// Mitsubishi GX Works2 project: 02.CumLongVo   PLC: FX3U/FX3UC

// global labels: Positon
VAR_GLOBAL
  Ser_Org : BOOL;
  Ser_Home_Done : BOOL;
  A_M : BOOL;
  Emer : BOOL;
  ON_ABS : BOOL;
  Pos_Tag_ABS : DINT;  (* mm *)
  Speed_Tag_ABS : DINT;  (* mm/s *)
  Excute_ABS : BOOL;
END_VAR

// global labels: Pro_Con_TF_J
VAR_GLOBAL
  Rev_J_Done : BOOL;
  Pro_Rev_J : BOOL;
  Req_Cov_W_Rev : BOOL;
  Conv_TF_J_Ready : BOOL;
  D_Step3_TF_Frame : TIMER;
  Cf_Install_Frame : BOOL;
END_VAR

// global labels: Pro_Con_Wait
VAR_GLOBAL
  Conv_W_Ready : BOOL;
  Conv_W_Rev_Done : BOOL;
  Req_Clus_Ep_Rev : BOOL;
  D_Req_ClusEp_Rev : TIMER;
END_VAR

// global labels: Cluster_BT
VAR_GLOBAL
  BT_Req_Rev_J : BOOL;
END_VAR

// global labels: Pro_Clus_Ep
VAR_GLOBAL
  Clus_Ep_Ready_Rev : BOOL;
  Clus_Ep_Rev_Done : BOOL;
  Req_Con_Out_Rev : BOOL;
  Clus_Ep_Safety : BOOL;
  Ex_Ep_Frame : BOOL;
  Stp_Ep_Fr : INT;
  Pos_Saf : REAL;
  Pos_Kep : REAL;
  Pos_Ep : REAL;
  Pos_Tar : REAL;
  Ep_Done : BOOL;
  Pos_Safe_Cyl_DT : REAL;
END_VAR

// global labels: Pro_Conv_Out
VAR_GLOBAL
  Conv_Out_Ready_Rev : BOOL;
  Conv_Out_Rev_Done : BOOL;
  Req_Clus_Drill_Rev : BOOL;
  TimeOut_BT : TIMER;
  Stp_Measuse : INT;
  T_Val_Err_Ams : REAL;
  Val_Err_Ams : REAL;
  Result : INT;
  D_Measure : TIMER;
  Stp_Rev_Conv_Out : BOOL;
  Measure_Done : BOOL;
  D_Conv_Out_Ready : TIMER;
  Standar_P : REAL;
  Standar_N : REAL;
  Value_1 : REAL;
  Value_2 : REAL;
  Value_Temp : REAL;
  D_Value2 : TIMER;
  Value_TempOut : REAL;
  O_Val_Err_Ams : REAL;
END_VAR

// global labels: TF_Jig
VAR_GLOBAL
  Step_TF_J : INT;
  Ex_TF_J : BOOL;
  Done_TF_J : BOOL;
  D_Done_J : TIMER;
END_VAR

// global labels: Clus_Drill
VAR_GLOBAL
  Clus_Drill_Ready_Rev : BOOL;
END_VAR

// global labels: Pro_Clus_TF_Frame
VAR_GLOBAL
  Clus_Cyl_TF_Frame_Ready : BOOL;  (* Ready *)
  Ex_TF_Frame : BOOL;
  D_Noti_Ex_Ep : TIMER;
  D_Nha_Kep1 : TIMER;
  D_PickDone : TIMER;
  Skip_Heater : BOOL;
  Stp_TF_Fr : INT;
  Clus_TF_Frame_Safety : BOOL;
  Ready_TF_Frame : BOOL;
  TF_Frame_Safe_Ep : BOOL;
  TF_Fr_Codition_TF_J : BOOL;
END_VAR

// global labels: Pro_Heater
VAR_GLOBAL
  Ex_Heater : BOOL;
  Heater_Done : BOOL;
  Heater_Busy : BOOL;
  Heater_Ready : BOOL;
  Heater_Safety : BOOL;
  Stp_Heater : INT;
  T_Target : REAL;
  Pre_Heater : BOOL;
END_VAR

PROGRAM Main
VAR
  Conv_TF_J : Conv_TF_J;
  Conv_Wait : Conv_Wait;
  C_Cyl_TF_J : C_Cyl_TF_J;
  C_Cyl_TF_SP : C_Cyl_TF_SP;
  Heater : Heater;
  Conv_Out : Conv_Out;
  Ctr_Mc : Ctr_MC;
  C_Shell : C_ShellCage;
END_VAR
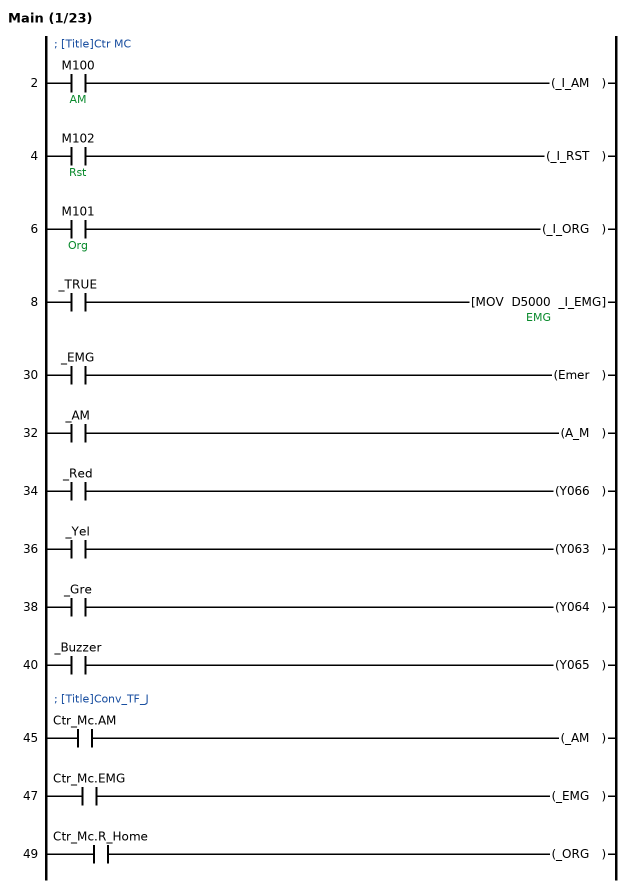
; FB BLK START Ctr_MC(Ctr_Mc)
; [Title]Ctr MC
2     LD      M100  ; AM
      OUT     _I_AM
4     LD      M102  ; Rst
      OUT     _I_RST
6     LD      M101  ; Org
      OUT     _I_ORG
8     LD      _TRUE
      MOV     D5000 _I_EMG  ; EMG
; FB START
; FB_NAME Ctr_MC
; INSTANCE_NAME Ctr_Mc
; FB IN_B:I_AM
; FB OUT_Flag_Run:B
; FB IN_B:I_RST
; FB OUT_EMG:B
; FB IN_B:I_ORG
; FB OUT_AM:B
; FB IN_W:I_EMG
; FB OUT_R_Home:B
; FB OUT_Red:B
; FB OUT_Yel:B
; FB OUT_Gre:B
; FB OUT_Buzzer:B
; FB END
30    LD      _EMG
      OUT     Emer
32    LD      _AM
      OUT     A_M
34    LD      _Red
      OUT     Y066
36    LD      _Yel
      OUT     Y063
38    LD      _Gre
      OUT     Y064
40    LD      _Buzzer
      OUT     Y065
; FB BLK END
; FB BLK START Conv_TF_J(Conv_TF_J)
; [Title]Conv_TF_J
45    LD      Ctr_Mc.AM
      OUT     _AM
47    LD      Ctr_Mc.EMG
      OUT     _EMG
49    LD      Ctr_Mc.R_Home
      OUT     _ORG
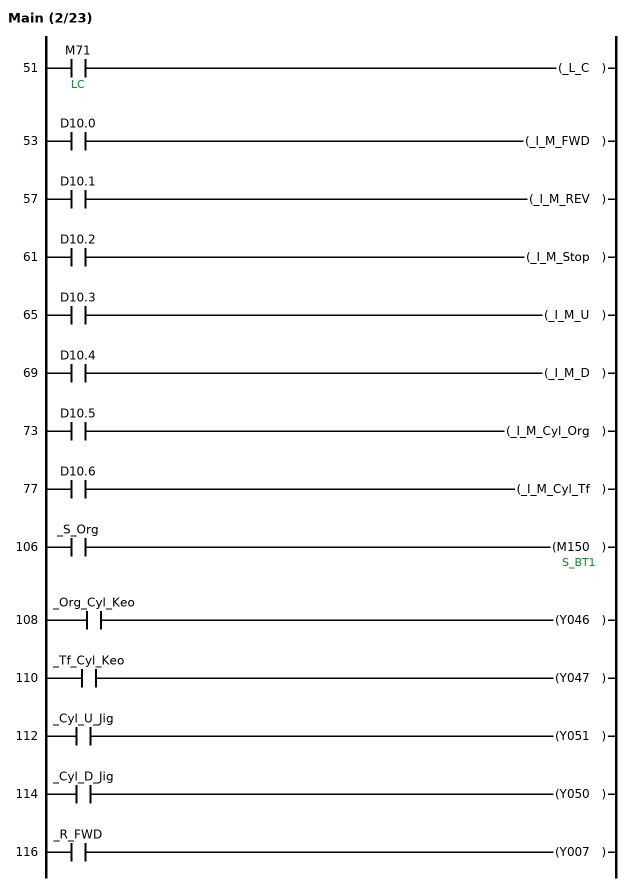
51    LD      M71  ; LC
      OUT     _L_C
53    LD      D10.0
      OUT     _I_M_FWD
57    LD      D10.1
      OUT     _I_M_REV
61    LD      D10.2
      OUT     _I_M_Stop
65    LD      D10.3
      OUT     _I_M_U
69    LD      D10.4
      OUT     _I_M_D
73    LD      D10.5
      OUT     _I_M_Cyl_Org
77    LD      D10.6
      OUT     _I_M_Cyl_Tf
; FB START
; FB_NAME Conv_TF_J
; INSTANCE_NAME Conv_TF_J
; FB IN_B:AM
; FB OUT_S_Org:B
; FB IN_B:EMG
; FB OUT_Org_Cyl_Keo:B
; FB IN_B:ORG
; FB OUT_Tf_Cyl_Keo:B
; FB IN_B:L_C
; FB OUT_Cyl_U_Jig:B
; FB IN_B:I_M_FWD
; FB OUT_Cyl_D_Jig:B
; FB IN_B:I_M_REV
; FB OUT_R_FWD:B
; FB IN_B:I_M_Stop
; FB OUT_R_REV:B
; FB IN_B:I_M_U
; FB IN_B:I_M_D
; FB IN_B:I_M_Cyl_Org
; FB IN_B:I_M_Cyl_Tf
; FB IN_W:A_S_Cyl_UD
; FB IN_W:A_S_Cyl_Tf
; FB IN_W:A_S_Conv
; FB END
106   LD      _S_Org
      OUT     M150  ; S_BT1
108   LD      _Org_Cyl_Keo
      OUT     Y046
110   LD      _Tf_Cyl_Keo
      OUT     Y047
112   LD      _Cyl_U_Jig
      OUT     Y051
114   LD      _Cyl_D_Jig
      OUT     Y050
116   LD      _R_FWD
      OUT     Y007
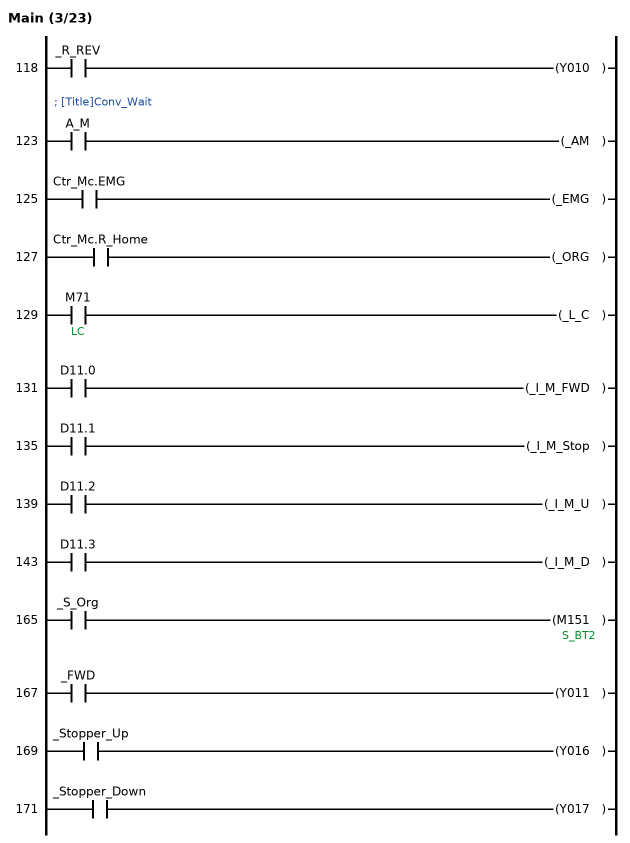
118   LD      _R_REV
      OUT     Y010
; FB BLK END
; FB BLK START Conv_Wait(Conv_Wait)
; [Title]Conv_Wait
123   LD      A_M
      OUT     _AM
125   LD      Ctr_Mc.EMG
      OUT     _EMG
127   LD      Ctr_Mc.R_Home
      OUT     _ORG
129   LD      M71  ; LC
      OUT     _L_C
131   LD      D11.0
      OUT     _I_M_FWD
135   LD      D11.1
      OUT     _I_M_Stop
139   LD      D11.2
      OUT     _I_M_U
143   LD      D11.3
      OUT     _I_M_D
; FB START
; FB_NAME Conv_Wait
; INSTANCE_NAME Conv_Wait
; FB IN_B:AM
; FB OUT_S_Org:B
; FB IN_B:EMG
; FB OUT_FWD:B
; FB IN_B:ORG
; FB OUT_Stopper_Up:B
; FB IN_B:L_C
; FB OUT_Stopper_Down:B
; FB IN_B:I_M_FWD
; FB IN_B:I_M_Stop
; FB IN_B:I_M_U
; FB IN_B:I_M_D
; FB IN_B:A_FWD
; FB IN_W:A_S_Stp
; FB END
165   LD      _S_Org
      OUT     M151  ; S_BT2
167   LD      _FWD
      OUT     Y011
169   LD      _Stopper_Up
      OUT     Y016
171   LD      _Stopper_Down
      OUT     Y017
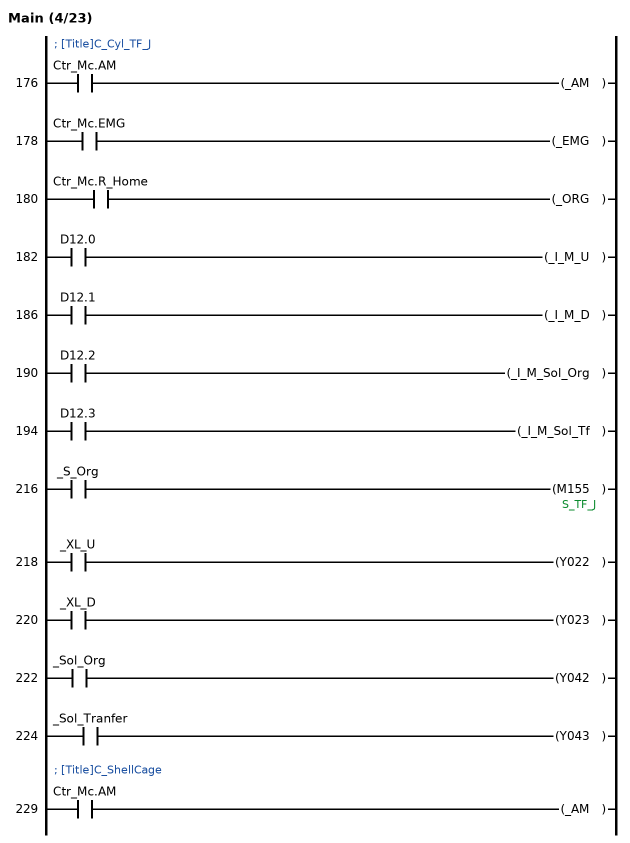
; FB BLK END
; FB BLK START C_Cyl_TF_J(C_Cyl_TF_J)
; [Title]C_Cyl_TF_J
176   LD      Ctr_Mc.AM
      OUT     _AM
178   LD      Ctr_Mc.EMG
      OUT     _EMG
180   LD      Ctr_Mc.R_Home
      OUT     _ORG
182   LD      D12.0
      OUT     _I_M_U
186   LD      D12.1
      OUT     _I_M_D
190   LD      D12.2
      OUT     _I_M_Sol_Org
194   LD      D12.3
      OUT     _I_M_Sol_Tf
; FB START
; FB_NAME C_Cyl_TF_J
; INSTANCE_NAME C_Cyl_TF_J
; FB IN_B:AM
; FB OUT_S_Org:B
; FB IN_B:EMG
; FB OUT_XL_U:B
; FB IN_B:ORG
; FB OUT_XL_D:B
; FB IN_B:I_M_U
; FB OUT_Sol_Org:B
; FB IN_B:I_M_D
; FB OUT_Sol_Tranfer:B
; FB IN_B:I_M_Sol_Org
; FB IN_B:I_M_Sol_Tf
; FB IN_W:A_Status_XL_U
; FB IN_W:A_S_Cyl_Tf
; FB END
216   LD      _S_Org
      OUT     M155  ; S_TF_J
218   LD      _XL_U
      OUT     Y022
220   LD      _XL_D
      OUT     Y023
222   LD      _Sol_Org
      OUT     Y042
224   LD      _Sol_Tranfer
      OUT     Y043
; FB BLK END
; FB BLK START C_ShellCage(C_Shell)
; [Title]C_ShellCage
229   LD      Ctr_Mc.AM
      OUT     _AM
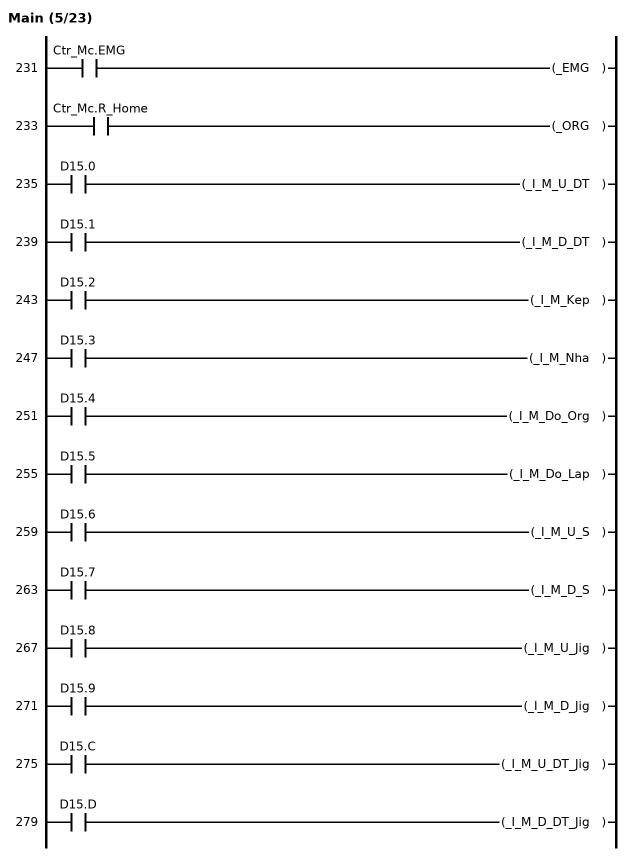
231   LD      Ctr_Mc.EMG
      OUT     _EMG
233   LD      Ctr_Mc.R_Home
      OUT     _ORG
235   LD      D15.0
      OUT     _I_M_U_DT
239   LD      D15.1
      OUT     _I_M_D_DT
243   LD      D15.2
      OUT     _I_M_Kep
247   LD      D15.3
      OUT     _I_M_Nha
251   LD      D15.4
      OUT     _I_M_Do_Org
255   LD      D15.5
      OUT     _I_M_Do_Lap
259   LD      D15.6
      OUT     _I_M_U_S
263   LD      D15.7
      OUT     _I_M_D_S
267   LD      D15.8
      OUT     _I_M_U_Jig
271   LD      D15.9
      OUT     _I_M_D_Jig
275   LD      D15.C
      OUT     _I_M_U_DT_Jig
279   LD      D15.D
      OUT     _I_M_D_DT_Jig
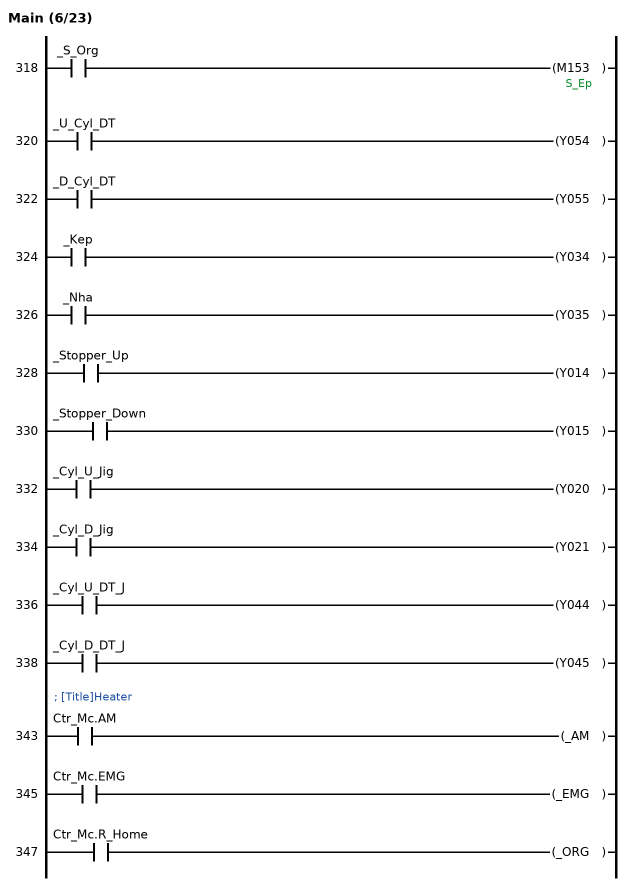
; FB START
; FB_NAME C_ShellCage
; INSTANCE_NAME C_Shell
; FB IN_B:AM
; FB OUT_S_Org:B
; FB IN_B:EMG
; FB OUT_U_Cyl_DT:B
; FB IN_B:ORG
; FB OUT_D_Cyl_DT:B
; FB IN_B:I_M_U_DT
; FB OUT_Kep:B
; FB IN_B:I_M_D_DT
; FB OUT_Nha:B
; FB IN_B:I_M_Kep
; FB OUT_Stopper_Up:B
; FB IN_B:I_M_Nha
; FB OUT_Stopper_Down:B
; FB IN_B:I_M_Do_Org
; FB OUT_Cyl_U_Jig:B
; FB IN_B:I_M_Do_Lap
; FB OUT_Cyl_D_Jig:B
; FB IN_B:I_M_U_S
; FB OUT_Cyl_U_DT_J:B
; FB IN_B:I_M_D_S
; FB OUT_Cyl_D_DT_J:B
; FB IN_B:I_M_U_Jig
; FB IN_B:I_M_D_Jig
; FB IN_B:I_M_U_DT_Jig
; FB IN_B:I_M_D_DT_Jig
; FB IN_W:A_S_Cyl_DT
; FB IN_W:A_S_Cyl_Kep
; FB IN_W:A_S_Stp
; FB IN_W:A_S_UD_J
; FB IN_W:A_S_DT_J
; FB END
318   LD      _S_Org
      OUT     M153  ; S_Ep
320   LD      _U_Cyl_DT
      OUT     Y054
322   LD      _D_Cyl_DT
      OUT     Y055
324   LD      _Kep
      OUT     Y034
326   LD      _Nha
      OUT     Y035
328   LD      _Stopper_Up
      OUT     Y014
330   LD      _Stopper_Down
      OUT     Y015
332   LD      _Cyl_U_Jig
      OUT     Y020
334   LD      _Cyl_D_Jig
      OUT     Y021
336   LD      _Cyl_U_DT_J
      OUT     Y044
338   LD      _Cyl_D_DT_J
      OUT     Y045
; FB BLK END
; FB BLK START Heater(Heater)
; [Title]Heater
343   LD      Ctr_Mc.AM
      OUT     _AM
345   LD      Ctr_Mc.EMG
      OUT     _EMG
347   LD      Ctr_Mc.R_Home
      OUT     _ORG
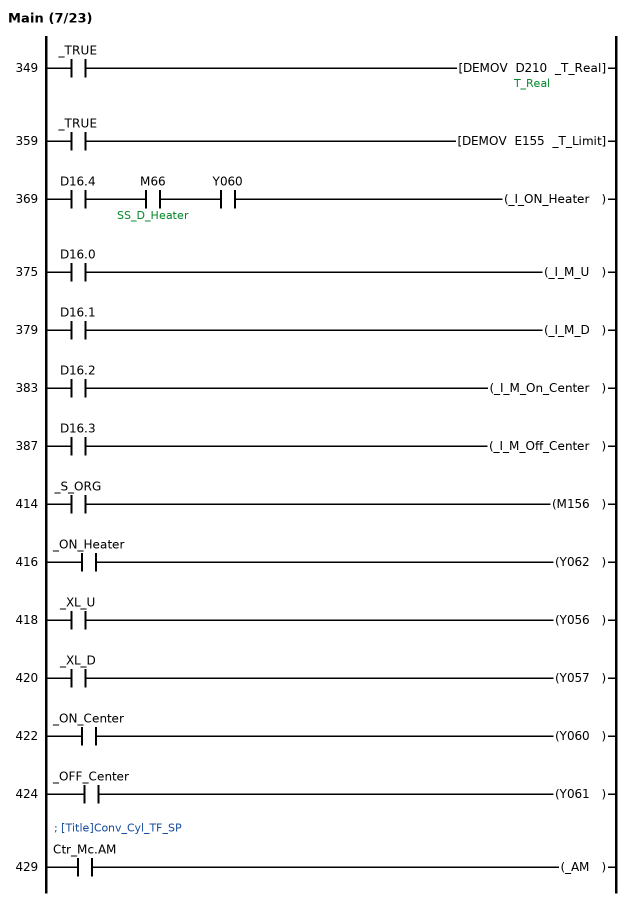
349   LD      _TRUE
      DEMOV   D210 _T_Real  ; T_Real
359   LD      _TRUE
      DEMOV   E155 _T_Limit
369   LD      D16.4
      AND     M66  ; SS_D_Heater
      AND     Y060
      OUT     _I_ON_Heater
375   LD      D16.0
      OUT     _I_M_U
379   LD      D16.1
      OUT     _I_M_D
383   LD      D16.2
      OUT     _I_M_On_Center
387   LD      D16.3
      OUT     _I_M_Off_Center
; FB START
; FB_NAME Heater
; INSTANCE_NAME Heater
; FB IN_B:AM
; FB OUT_S_ORG:B
; FB IN_B:EMG
; FB OUT_ON_Heater:B
; FB IN_B:ORG
; FB OUT_XL_U:B
; FB IN_E:T_Real
; FB OUT_XL_D:B
; FB IN_E:T_Limit
; FB OUT_ON_Center:B
; FB IN_B:I_ON_Heater
; FB OUT_OFF_Center:B
; FB IN_B:I_M_U
; FB IN_B:I_M_D
; FB IN_B:I_M_On_Center
; FB IN_B:I_M_Off_Center
; FB IN_B:A_ON_Heater
; FB IN_W:A_S_Cyl_UD
; FB IN_W:A_Status_Center
; FB END
414   LD      _S_ORG
      OUT     M156
416   LD      _ON_Heater
      OUT     Y062
418   LD      _XL_U
      OUT     Y056
420   LD      _XL_D
      OUT     Y057
422   LD      _ON_Center
      OUT     Y060
424   LD      _OFF_Center
      OUT     Y061
; FB BLK END
; FB BLK START C_Cyl_TF_SP(C_Cyl_TF_SP)
; [Title]Conv_Cyl_TF_SP
429   LD      Ctr_Mc.AM
      OUT     _AM
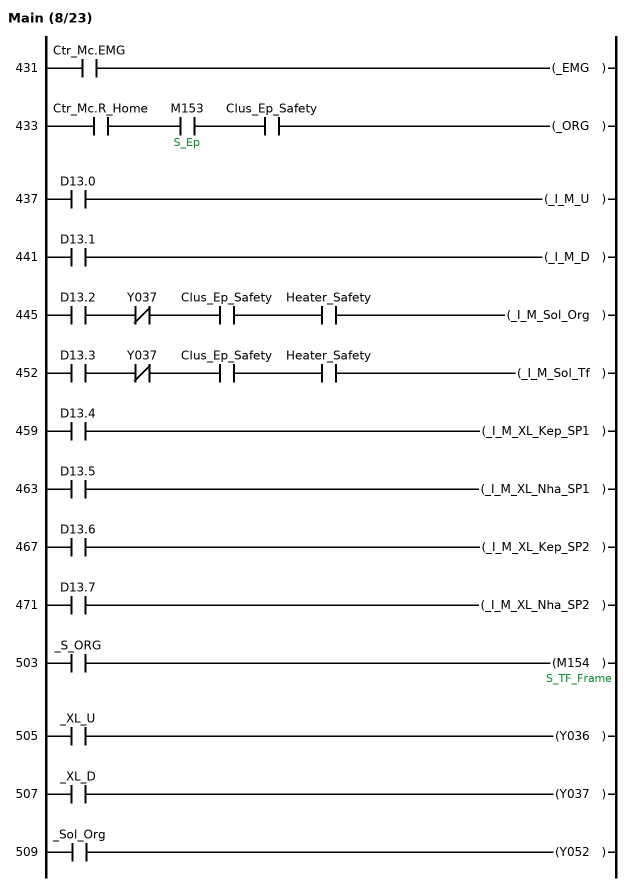
431   LD      Ctr_Mc.EMG
      OUT     _EMG
433   LD      Ctr_Mc.R_Home
      AND     M153  ; S_Ep
      AND     Clus_Ep_Safety
      OUT     _ORG
437   LD      D13.0
      OUT     _I_M_U
441   LD      D13.1
      OUT     _I_M_D
445   LD      D13.2
      ANI     Y037
      AND     Clus_Ep_Safety
      AND     Heater_Safety
      OUT     _I_M_Sol_Org
452   LD      D13.3
      ANI     Y037
      AND     Clus_Ep_Safety
      AND     Heater_Safety
      OUT     _I_M_Sol_Tf
459   LD      D13.4
      OUT     _I_M_XL_Kep_SP1
463   LD      D13.5
      OUT     _I_M_XL_Nha_SP1
467   LD      D13.6
      OUT     _I_M_XL_Kep_SP2
471   LD      D13.7
      OUT     _I_M_XL_Nha_SP2
; FB START
; FB_NAME C_Cyl_TF_SP
; INSTANCE_NAME C_Cyl_TF_SP
; FB IN_B:AM
; FB OUT_S_ORG:B
; FB IN_B:EMG
; FB OUT_XL_U:B
; FB IN_B:ORG
; FB OUT_XL_D:B
; FB IN_B:I_M_U
; FB OUT_Sol_Org:B
; FB IN_B:I_M_D
; FB OUT_Sol_Tranfer:B
; FB IN_B:I_M_Sol_Org
; FB OUT_XL_Kep_SP1:B
; FB IN_B:I_M_Sol_Tf
; FB OUT_XL_Mo_SP1:B
; FB IN_B:I_M_XL_Kep_SP1
; FB OUT_XL_Kep_SP2:B
; FB IN_B:I_M_XL_Nha_SP1
; FB OUT_XL_Mo_SP2:B
; FB IN_B:I_M_XL_Kep_SP2
; FB IN_B:I_M_XL_Nha_SP2
; FB IN_W:A_Status_XL_U
; FB IN_W:A_S_Cyl_Tf
; FB IN_W:A_S_Cyl_Kep_1
; FB IN_W:A_S_Cyl_Kep_2
; FB END
503   LD      _S_ORG
      OUT     M154  ; S_TF_Frame
505   LD      _XL_U
      OUT     Y036
507   LD      _XL_D
      OUT     Y037
509   LD      _Sol_Org
      OUT     Y052
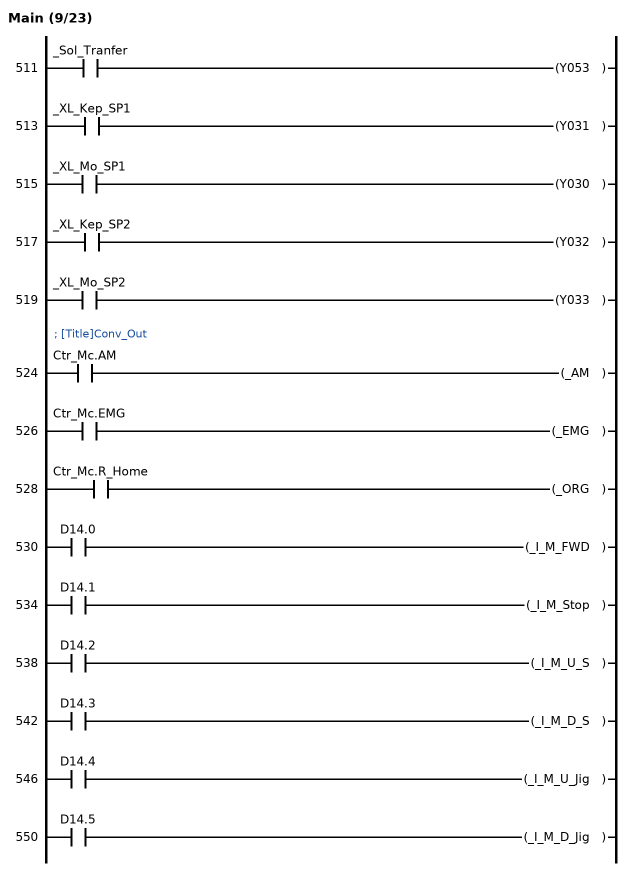
511   LD      _Sol_Tranfer
      OUT     Y053
513   LD      _XL_Kep_SP1
      OUT     Y031
515   LD      _XL_Mo_SP1
      OUT     Y030
517   LD      _XL_Kep_SP2
      OUT     Y032
519   LD      _XL_Mo_SP2
      OUT     Y033
; FB BLK END
; FB BLK START Conv_Out(Conv_Out)
; [Title]Conv_Out
524   LD      Ctr_Mc.AM
      OUT     _AM
526   LD      Ctr_Mc.EMG
      OUT     _EMG
528   LD      Ctr_Mc.R_Home
      OUT     _ORG
530   LD      D14.0
      OUT     _I_M_FWD
534   LD      D14.1
      OUT     _I_M_Stop
538   LD      D14.2
      OUT     _I_M_U_S
542   LD      D14.3
      OUT     _I_M_D_S
546   LD      D14.4
      OUT     _I_M_U_Jig
550   LD      D14.5
      OUT     _I_M_D_Jig
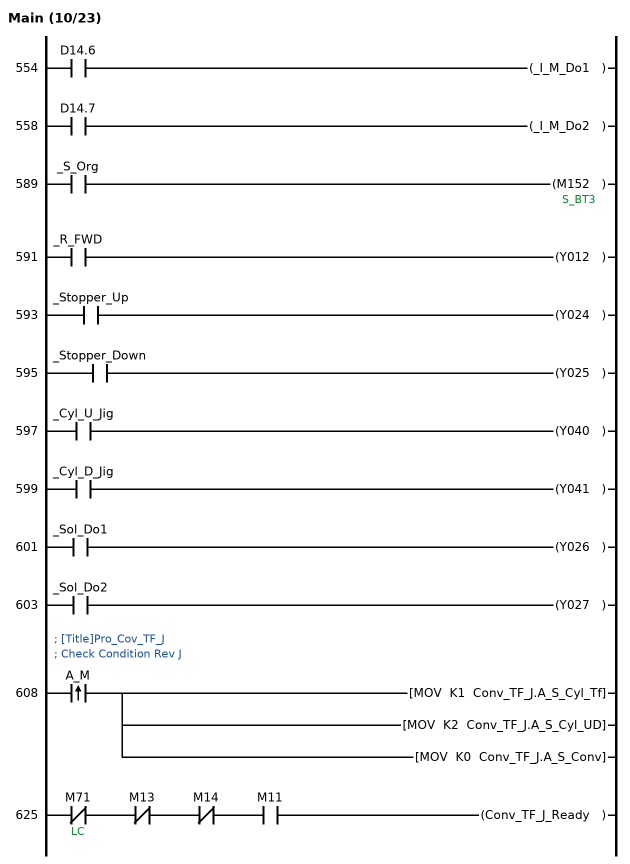
554   LD      D14.6
      OUT     _I_M_Do1
558   LD      D14.7
      OUT     _I_M_Do2
; FB START
; FB_NAME Conv_Out
; INSTANCE_NAME Conv_Out
; FB IN_B:AM
; FB OUT_S_Org:B
; FB IN_B:EMG
; FB OUT_R_FWD:B
; FB IN_B:ORG
; FB OUT_Stopper_Up:B
; FB IN_B:I_M_FWD
; FB OUT_Stopper_Down:B
; FB IN_B:I_M_Stop
; FB OUT_Cyl_U_Jig:B
; FB IN_B:I_M_U_S
; FB OUT_Cyl_D_Jig:B
; FB IN_B:I_M_D_S
; FB OUT_Sol_Do1:B
; FB IN_B:I_M_U_Jig
; FB OUT_Sol_Do2:B
; FB IN_B:I_M_D_Jig
; FB IN_B:I_M_Do1
; FB IN_B:I_M_Do2
; FB IN_W:A_S_Cyl_UD
; FB IN_W:A_S_Stp
; FB IN_B:A_FWD
; FB IN_W:A_S_Do
; FB END
589   LD      _S_Org
      OUT     M152  ; S_BT3
591   LD      _R_FWD
      OUT     Y012
593   LD      _Stopper_Up
      OUT     Y024
595   LD      _Stopper_Down
      OUT     Y025
597   LD      _Cyl_U_Jig
      OUT     Y040
599   LD      _Cyl_D_Jig
      OUT     Y041
601   LD      _Sol_Do1
      OUT     Y026
603   LD      _Sol_Do2
      OUT     Y027
; FB BLK END
; [Title]Pro_Cov_TF_J
; Check Condition Rev J
608   LDP     A_M
      MOV     K1 Conv_TF_J.A_S_Cyl_Tf
      MOV     K2 Conv_TF_J.A_S_Cyl_UD
      MOV     K0 Conv_TF_J.A_S_Conv
625   LDI     M71  ; LC
      ANI     M13
      ANI     M14
      AND     M11
      OUT     Conv_TF_J_Ready
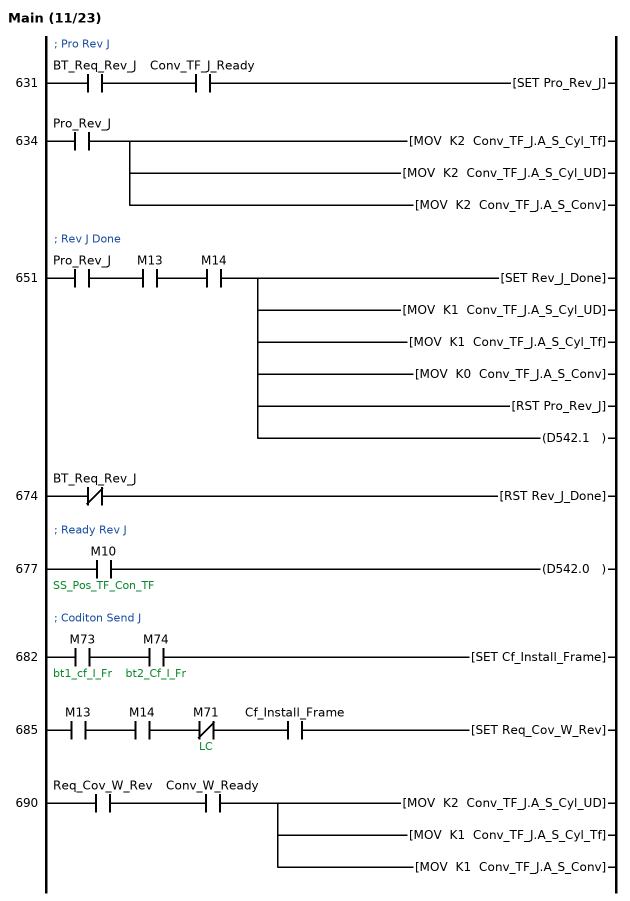
; Pro Rev J
631   LD      BT_Req_Rev_J
      AND     Conv_TF_J_Ready
      SET     Pro_Rev_J
634   LD      Pro_Rev_J
      MOV     K2 Conv_TF_J.A_S_Cyl_Tf
      MOV     K2 Conv_TF_J.A_S_Cyl_UD
      MOV     K2 Conv_TF_J.A_S_Conv
; Rev J Done
651   LD      Pro_Rev_J
      AND     M13
      AND     M14
      SET     Rev_J_Done
      MOV     K1 Conv_TF_J.A_S_Cyl_UD
      MOV     K1 Conv_TF_J.A_S_Cyl_Tf
      MOV     K0 Conv_TF_J.A_S_Conv
      RST     Pro_Rev_J
      OUT     D542.1
674   LDI     BT_Req_Rev_J
      RST     Rev_J_Done
; Ready Rev J
677   LD      M10  ; SS_Pos_TF_Con_TF
      OUT     D542.0
; Coditon Send J
682   LD      M73  ; bt1_cf_I_Fr
      AND     M74  ; bt2_Cf_I_Fr
      SET     Cf_Install_Frame
685   LD      M13
      AND     M14
      ANI     M71  ; LC
      AND     Cf_Install_Frame
      SET     Req_Cov_W_Rev
690   LD      Req_Cov_W_Rev
      AND     Conv_W_Ready
      MOV     K2 Conv_TF_J.A_S_Cyl_UD
      MOV     K1 Conv_TF_J.A_S_Cyl_Tf
      MOV     K1 Conv_TF_J.A_S_Conv
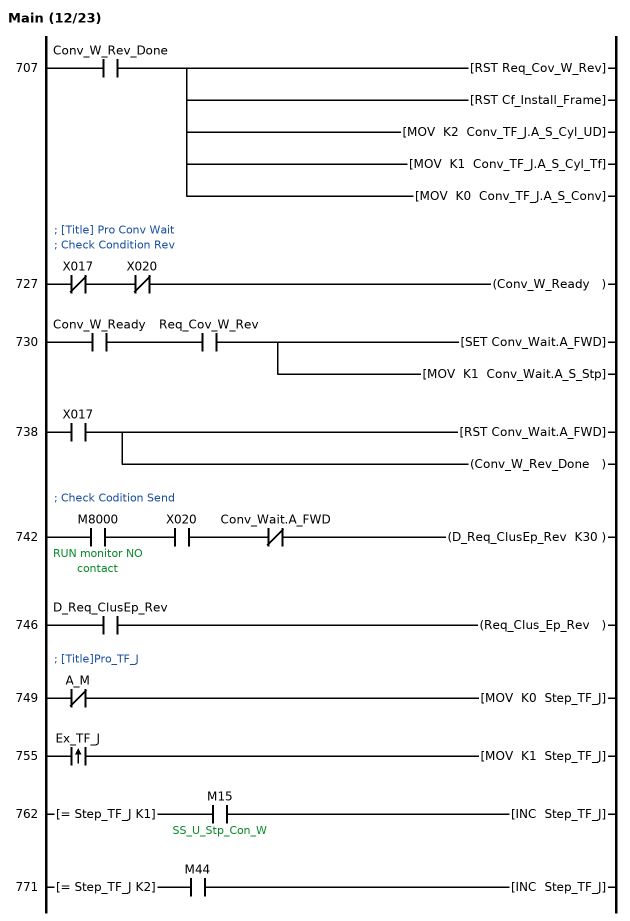
707   LD      Conv_W_Rev_Done
      RST     Req_Cov_W_Rev
      RST     Cf_Install_Frame
      MOV     K2 Conv_TF_J.A_S_Cyl_UD
      MOV     K1 Conv_TF_J.A_S_Cyl_Tf
      MOV     K0 Conv_TF_J.A_S_Conv
; [Title] Pro Conv Wait
; Check Condition Rev
727   LDI     X017
      ANI     X020
      OUT     Conv_W_Ready
730   LD      Conv_W_Ready
      AND     Req_Cov_W_Rev
      SET     Conv_Wait.A_FWD
      MOV     K1 Conv_Wait.A_S_Stp
738   LD      X017
      RST     Conv_Wait.A_FWD
      OUT     Conv_W_Rev_Done
; Check Codition Send
742   LD      M8000  ; RUN monitor NO contact
      AND     X020
      ANI     Conv_Wait.A_FWD
      OUT     D_Req_ClusEp_Rev K30
746   LD      D_Req_ClusEp_Rev
      OUT     Req_Clus_Ep_Rev
; [Title]Pro_TF_J
749   LDI     A_M
      MOV     K0 Step_TF_J
755   LDP     Ex_TF_J
      MOV     K1 Step_TF_J
762   LD=     Step_TF_J K1
      AND     M15  ; SS_U_Stp_Con_W
      INC     Step_TF_J
771   LD=     Step_TF_J K2
      AND     M44
      INC     Step_TF_J
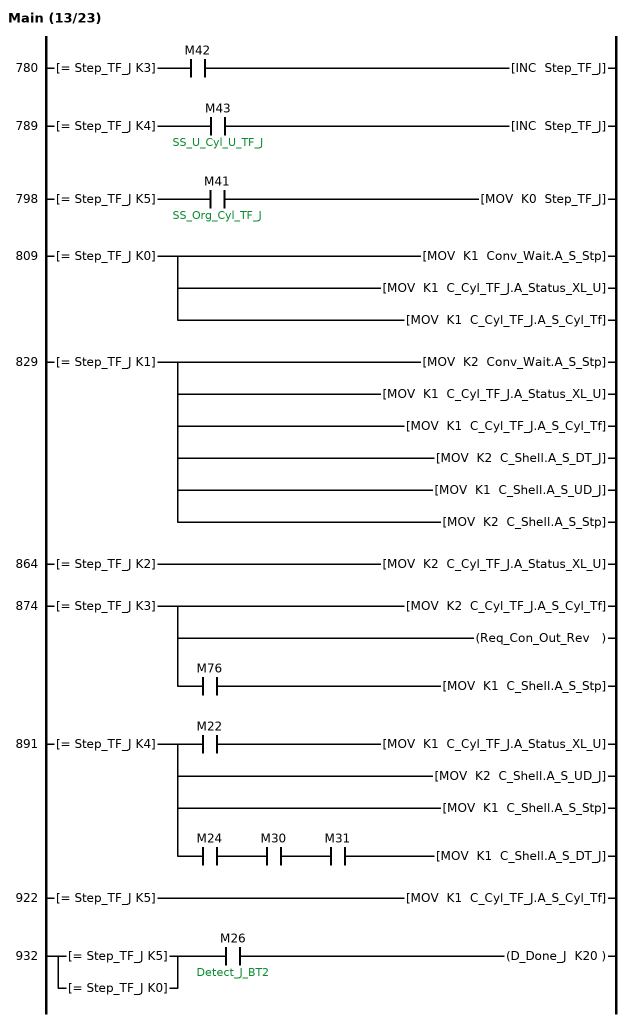
780   LD=     Step_TF_J K3
      AND     M42
      INC     Step_TF_J
789   LD=     Step_TF_J K4
      AND     M43  ; SS_U_Cyl_U_TF_J
      INC     Step_TF_J
798   LD=     Step_TF_J K5
      AND     M41  ; SS_Org_Cyl_TF_J
      MOV     K0 Step_TF_J
809   LD=     Step_TF_J K0
      MOV     K1 Conv_Wait.A_S_Stp
      MOV     K1 C_Cyl_TF_J.A_Status_XL_U
      MOV     K1 C_Cyl_TF_J.A_S_Cyl_Tf
829   LD=     Step_TF_J K1
      MOV     K2 Conv_Wait.A_S_Stp
      MOV     K1 C_Cyl_TF_J.A_Status_XL_U
      MOV     K1 C_Cyl_TF_J.A_S_Cyl_Tf
      MOV     K2 C_Shell.A_S_DT_J
      MOV     K1 C_Shell.A_S_UD_J
      MOV     K2 C_Shell.A_S_Stp
864   LD=     Step_TF_J K2
      MOV     K2 C_Cyl_TF_J.A_Status_XL_U
874   LD=     Step_TF_J K3
      MOV     K2 C_Cyl_TF_J.A_S_Cyl_Tf
      OUT     Req_Con_Out_Rev
      AND     M76
      MOV     K1 C_Shell.A_S_Stp
891   LD=     Step_TF_J K4
      MPS
      AND     M22
      MOV     K1 C_Cyl_TF_J.A_Status_XL_U
      MPP
      MOV     K2 C_Shell.A_S_UD_J
      MOV     K1 C_Shell.A_S_Stp
      AND     M24
      AND     M30
      AND     M31
      MOV     K1 C_Shell.A_S_DT_J
922   LD=     Step_TF_J K5
      MOV     K1 C_Cyl_TF_J.A_S_Cyl_Tf
932   LD=     Step_TF_J K5
      OR=     Step_TF_J K0
      AND     M26  ; Detect_J_BT2
      OUT     D_Done_J K20
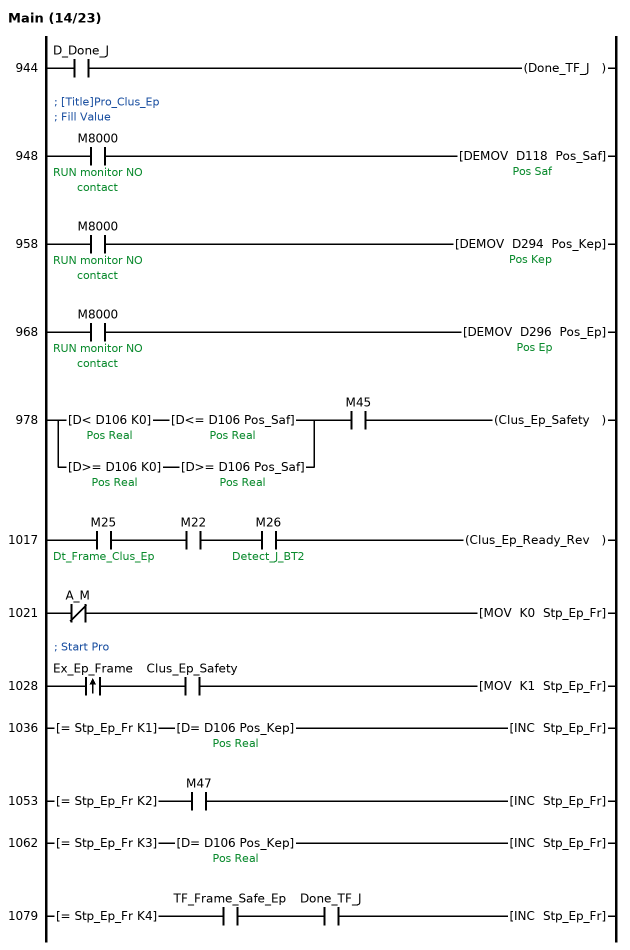
944   LD      D_Done_J
      OUT     Done_TF_J
; [Title]Pro_Clus_Ep
; Fill Value
948   LD      M8000  ; RUN monitor NO contact
      DEMOV   D118 Pos_Saf  ; Pos Saf
958   LD      M8000  ; RUN monitor NO contact
      DEMOV   D294 Pos_Kep  ; Pos Kep
968   LD      M8000  ; RUN monitor NO contact
      DEMOV   D296 Pos_Ep  ; Pos Ep
978   LDD<    D106 K0  ; Pos Real
      ANDD<=  D106 Pos_Saf  ; Pos Real
      LDD>=   D106 K0  ; Pos Real
      ANDD>=  D106 Pos_Saf  ; Pos Real
      ORB
      AND     M45
      OUT     Clus_Ep_Safety
1017  LD      M25  ; Dt_Frame_Clus_Ep
      AND     M22
      AND     M26  ; Detect_J_BT2
      OUT     Clus_Ep_Ready_Rev
1021  LDI     A_M
      MOV     K0 Stp_Ep_Fr
; Start Pro
1028  LDP     Ex_Ep_Frame
      AND     Clus_Ep_Safety
      MOV     K1 Stp_Ep_Fr
1036  LD=     Stp_Ep_Fr K1
      ANDD=   D106 Pos_Kep  ; Pos Real
      INC     Stp_Ep_Fr
1053  LD=     Stp_Ep_Fr K2
      AND     M47
      INC     Stp_Ep_Fr
1062  LD=     Stp_Ep_Fr K3
      ANDD=   D106 Pos_Kep  ; Pos Real
      INC     Stp_Ep_Fr
1079  LD=     Stp_Ep_Fr K4
      AND     TF_Frame_Safe_Ep
      AND     Done_TF_J
      INC     Stp_Ep_Fr
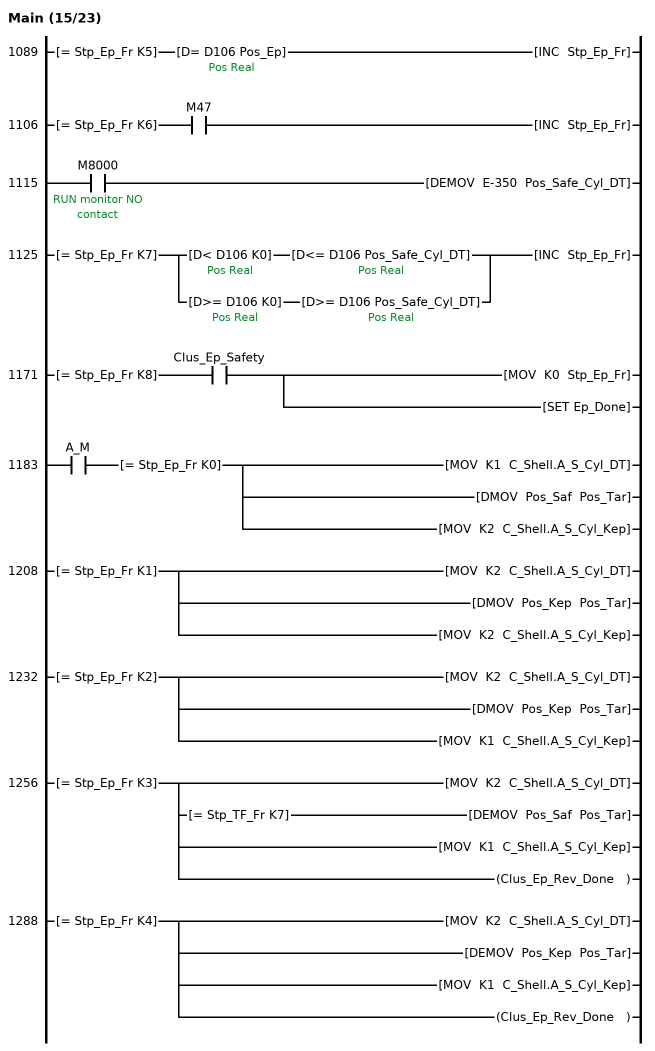
1089  LD=     Stp_Ep_Fr K5
      ANDD=   D106 Pos_Ep  ; Pos Real
      INC     Stp_Ep_Fr
1106  LD=     Stp_Ep_Fr K6
      AND     M47
      INC     Stp_Ep_Fr
1115  LD      M8000  ; RUN monitor NO contact
      DEMOV   E-350 Pos_Safe_Cyl_DT
1125  LD=     Stp_Ep_Fr K7
      LDD<    D106 K0  ; Pos Real
      ANDD<=  D106 Pos_Safe_Cyl_DT  ; Pos Real
      LDD>=   D106 K0  ; Pos Real
      ANDD>=  D106 Pos_Safe_Cyl_DT  ; Pos Real
      ORB
      ANB
      INC     Stp_Ep_Fr
1171  LD=     Stp_Ep_Fr K8
      AND     Clus_Ep_Safety
      MOV     K0 Stp_Ep_Fr
      SET     Ep_Done
1183  LD      A_M
      AND=    Stp_Ep_Fr K0
      MOV     K1 C_Shell.A_S_Cyl_DT
      DMOV    Pos_Saf Pos_Tar
      MOV     K2 C_Shell.A_S_Cyl_Kep
1208  LD=     Stp_Ep_Fr K1
      MOV     K2 C_Shell.A_S_Cyl_DT
      DMOV    Pos_Kep Pos_Tar
      MOV     K2 C_Shell.A_S_Cyl_Kep
1232  LD=     Stp_Ep_Fr K2
      MOV     K2 C_Shell.A_S_Cyl_DT
      DMOV    Pos_Kep Pos_Tar
      MOV     K1 C_Shell.A_S_Cyl_Kep
1256  LD=     Stp_Ep_Fr K3
      MOV     K2 C_Shell.A_S_Cyl_DT
      MPS
      AND=    Stp_TF_Fr K7
      DEMOV   Pos_Saf Pos_Tar
      MPP
      MOV     K1 C_Shell.A_S_Cyl_Kep
      OUT     Clus_Ep_Rev_Done
1288  LD=     Stp_Ep_Fr K4
      MOV     K2 C_Shell.A_S_Cyl_DT
      DEMOV   Pos_Kep Pos_Tar
      MOV     K1 C_Shell.A_S_Cyl_Kep
      OUT     Clus_Ep_Rev_Done
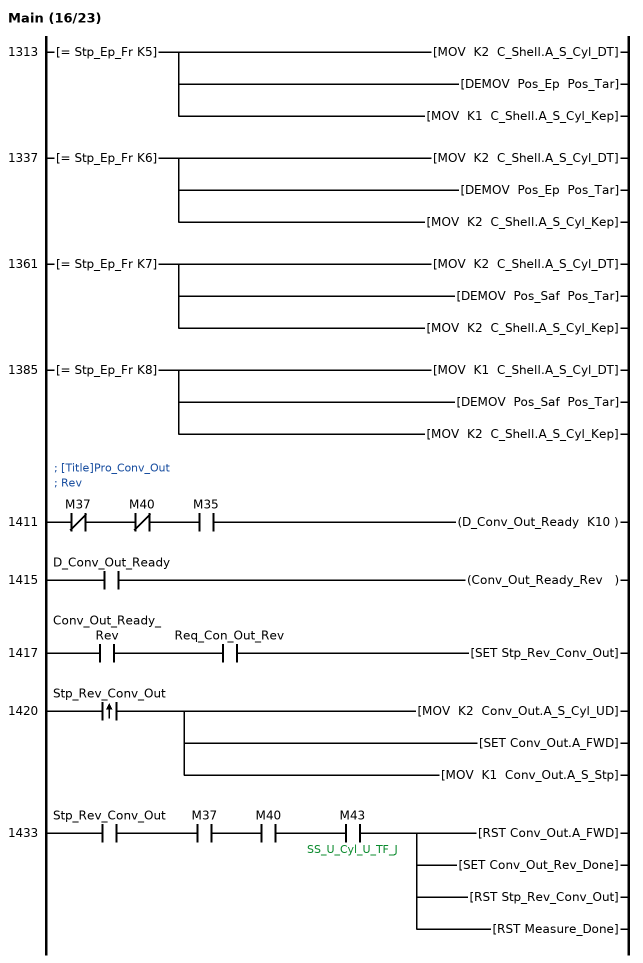
1313  LD=     Stp_Ep_Fr K5
      MOV     K2 C_Shell.A_S_Cyl_DT
      DEMOV   Pos_Ep Pos_Tar
      MOV     K1 C_Shell.A_S_Cyl_Kep
1337  LD=     Stp_Ep_Fr K6
      MOV     K2 C_Shell.A_S_Cyl_DT
      DEMOV   Pos_Ep Pos_Tar
      MOV     K2 C_Shell.A_S_Cyl_Kep
1361  LD=     Stp_Ep_Fr K7
      MOV     K2 C_Shell.A_S_Cyl_DT
      DEMOV   Pos_Saf Pos_Tar
      MOV     K2 C_Shell.A_S_Cyl_Kep
1385  LD=     Stp_Ep_Fr K8
      MOV     K1 C_Shell.A_S_Cyl_DT
      DEMOV   Pos_Saf Pos_Tar
      MOV     K2 C_Shell.A_S_Cyl_Kep
; [Title]Pro_Conv_Out
; Rev
1411  LDI     M37
      ANI     M40
      AND     M35
      OUT     D_Conv_Out_Ready K10
1415  LD      D_Conv_Out_Ready
      OUT     Conv_Out_Ready_Rev
1417  LD      Conv_Out_Ready_Rev
      AND     Req_Con_Out_Rev
      SET     Stp_Rev_Conv_Out
1420  LDP     Stp_Rev_Conv_Out
      MOV     K2 Conv_Out.A_S_Cyl_UD
      SET     Conv_Out.A_FWD
      MOV     K1 Conv_Out.A_S_Stp
1433  LD      Stp_Rev_Conv_Out
      AND     M37
      AND     M40
      AND     M43  ; SS_U_Cyl_U_TF_J
      RST     Conv_Out.A_FWD
      SET     Conv_Out_Rev_Done
      RST     Stp_Rev_Conv_Out
      RST     Measure_Done
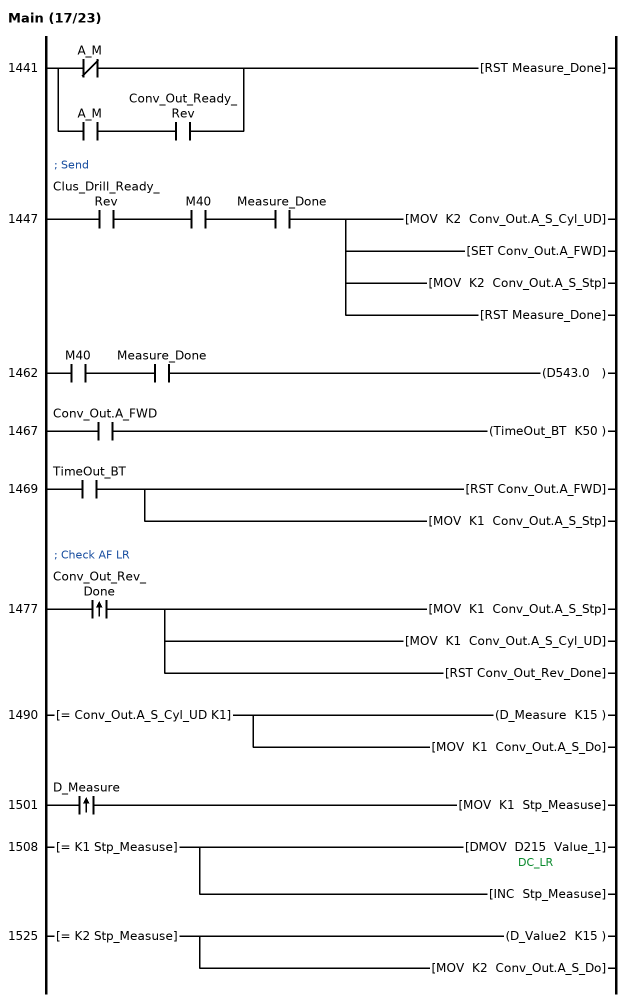
1441  LDI     A_M
      LD      A_M
      AND     Conv_Out_Ready_Rev
      ORB
      RST     Measure_Done
; Send
1447  LD      Clus_Drill_Ready_Rev
      AND     M40
      AND     Measure_Done
      MOV     K2 Conv_Out.A_S_Cyl_UD
      SET     Conv_Out.A_FWD
      MOV     K2 Conv_Out.A_S_Stp
      RST     Measure_Done
1462  LD      M40
      AND     Measure_Done
      OUT     D543.0
1467  LD      Conv_Out.A_FWD
      OUT     TimeOut_BT K50
1469  LD      TimeOut_BT
      RST     Conv_Out.A_FWD
      MOV     K1 Conv_Out.A_S_Stp
; Check AF LR
1477  LDP     Conv_Out_Rev_Done
      MOV     K1 Conv_Out.A_S_Stp
      MOV     K1 Conv_Out.A_S_Cyl_UD
      RST     Conv_Out_Rev_Done
1490  LD=     Conv_Out.A_S_Cyl_UD K1
      OUT     D_Measure K15
      MOV     K1 Conv_Out.A_S_Do
1501  LDP     D_Measure
      MOV     K1 Stp_Measuse
1508  LD=     K1 Stp_Measuse
      DMOV    D215 Value_1  ; DC_LR
      INC     Stp_Measuse
1525  LD=     K2 Stp_Measuse
      OUT     D_Value2 K15
      MOV     K2 Conv_Out.A_S_Do
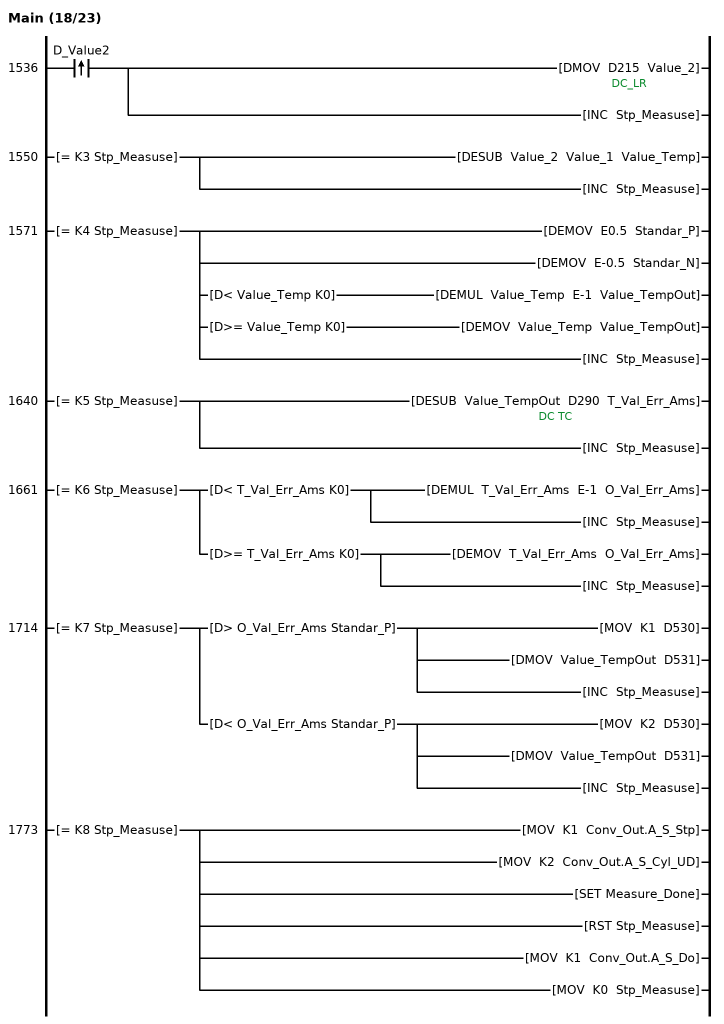
1536  LDP     D_Value2
      DMOV    D215 Value_2
      INC     Stp_Measuse
1550  LD=     K3 Stp_Measuse
      DESUB   Value_2 Value_1 Value_Temp
      INC     Stp_Measuse
1571  LD=     K4 Stp_Measuse
      DEMOV   E0.5 Standar_P
      DEMOV   E-0.5 Standar_N
      MPS
      ANDD<   Value_Temp K0
      DEMUL   Value_Temp E-1 Value_TempOut
      MRD
      ANDD>=  Value_Temp K0
      DEMOV   Value_Temp Value_TempOut
      MPP
      INC     Stp_Measuse
1640  LD=     K5 Stp_Measuse
      DESUB   Value_TempOut D290 T_Val_Err_Ams  ; DC TC
      INC     Stp_Measuse
1661  LD=     K6 Stp_Measuse
      MPS
      ANDD<   T_Val_Err_Ams K0
      DEMUL   T_Val_Err_Ams E-1 O_Val_Err_Ams
      INC     Stp_Measuse
      MPP
      ANDD>=  T_Val_Err_Ams K0
      DEMOV   T_Val_Err_Ams O_Val_Err_Ams
      INC     Stp_Measuse
1714  LD=     K7 Stp_Measuse
      MPS
      ANDD>   O_Val_Err_Ams Standar_P
      MOV     K1 D530
      DMOV    Value_TempOut D531
      INC     Stp_Measuse
      MPP
      ANDD<   O_Val_Err_Ams Standar_P
      MOV     K2 D530
      DMOV    Value_TempOut D531
      INC     Stp_Measuse
1773  LD=     K8 Stp_Measuse
      MOV     K1 Conv_Out.A_S_Stp
      MOV     K2 Conv_Out.A_S_Cyl_UD
      SET     Measure_Done
      RST     Stp_Measuse
      MOV     K1 Conv_Out.A_S_Do
      MOV     K0 Stp_Measuse
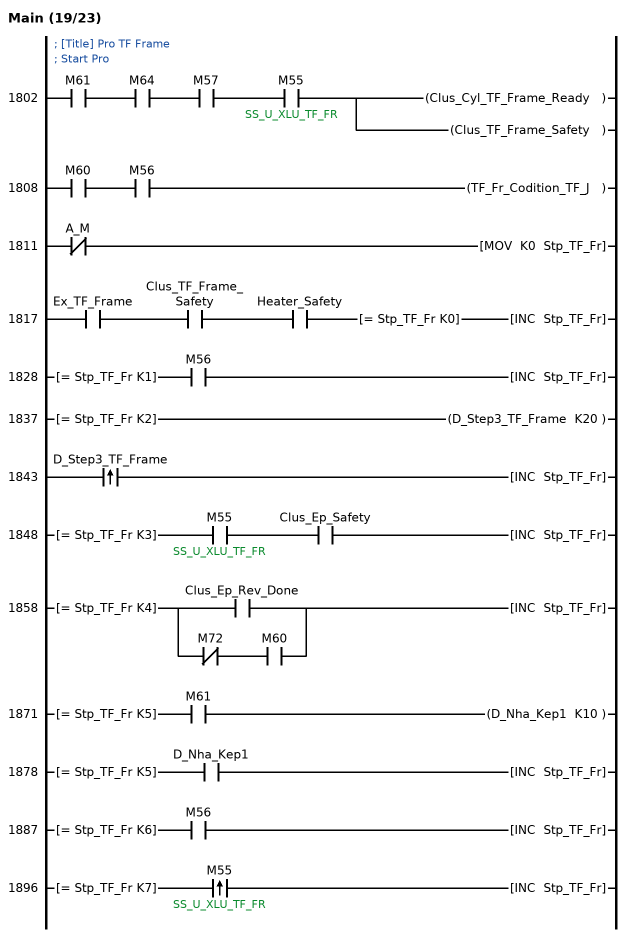
; [Title] Pro TF Frame
; Start Pro
1802  LD      M61
      AND     M64
      AND     M57
      AND     M55  ; SS_U_XLU_TF_FR
      OUT     Clus_Cyl_TF_Frame_Ready
      OUT     Clus_TF_Frame_Safety
1808  LD      M60
      AND     M56
      OUT     TF_Fr_Codition_TF_J
1811  LDI     A_M
      MOV     K0 Stp_TF_Fr
1817  LD      Ex_TF_Frame
      AND     Clus_TF_Frame_Safety
      AND     Heater_Safety
      AND=    Stp_TF_Fr K0
      INC     Stp_TF_Fr
1828  LD=     Stp_TF_Fr K1
      AND     M56
      INC     Stp_TF_Fr
1837  LD=     Stp_TF_Fr K2
      OUT     D_Step3_TF_Frame K20
1843  LDP     D_Step3_TF_Frame
      INC     Stp_TF_Fr
1848  LD=     Stp_TF_Fr K3
      AND     M55  ; SS_U_XLU_TF_FR
      AND     Clus_Ep_Safety
      INC     Stp_TF_Fr
1858  LD=     Stp_TF_Fr K4
      LD      Clus_Ep_Rev_Done
      LDI     M72
      AND     M60
      ORB
      ANB
      INC     Stp_TF_Fr
1871  LD=     Stp_TF_Fr K5
      AND     M61
      OUT     D_Nha_Kep1 K10
1878  LD=     Stp_TF_Fr K5
      AND     D_Nha_Kep1
      INC     Stp_TF_Fr
1887  LD=     Stp_TF_Fr K6
      AND     M56
      INC     Stp_TF_Fr
1896  LD=     Stp_TF_Fr K7
      ANDP    M55  ; SS_U_XLU_TF_FR
      INC     Stp_TF_Fr
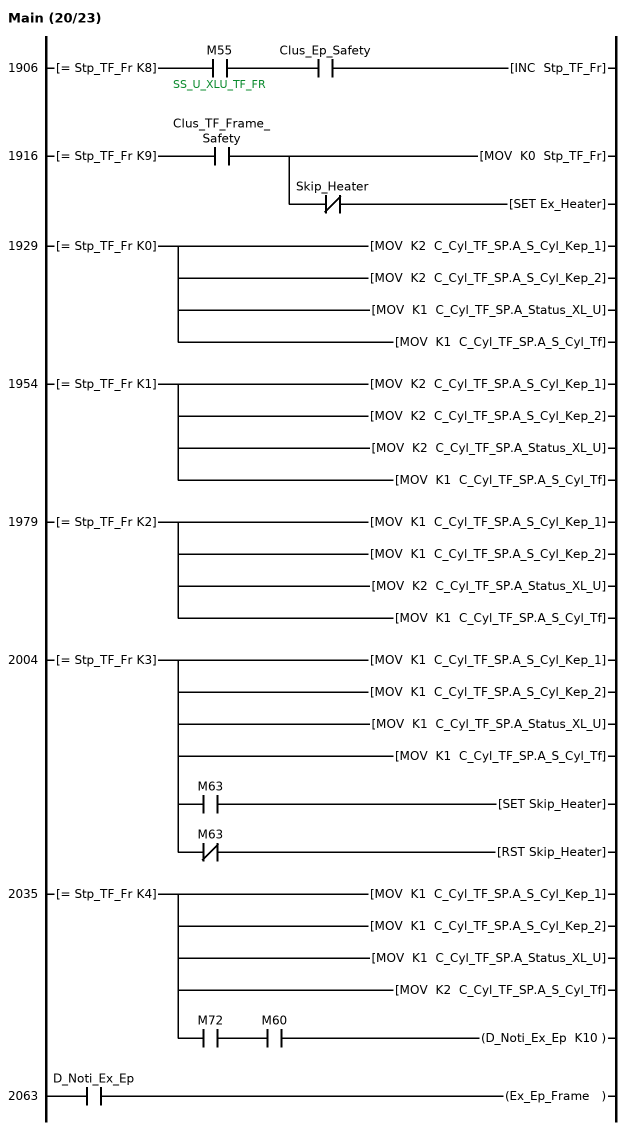
1906  LD=     Stp_TF_Fr K8
      AND     M55  ; SS_U_XLU_TF_FR
      AND     Clus_Ep_Safety
      INC     Stp_TF_Fr
1916  LD=     Stp_TF_Fr K9
      AND     Clus_TF_Frame_Safety
      MOV     K0 Stp_TF_Fr
      ANI     Skip_Heater
      SET     Ex_Heater
1929  LD=     Stp_TF_Fr K0
      MOV     K2 C_Cyl_TF_SP.A_S_Cyl_Kep_1
      MOV     K2 C_Cyl_TF_SP.A_S_Cyl_Kep_2
      MOV     K1 C_Cyl_TF_SP.A_Status_XL_U
      MOV     K1 C_Cyl_TF_SP.A_S_Cyl_Tf
1954  LD=     Stp_TF_Fr K1
      MOV     K2 C_Cyl_TF_SP.A_S_Cyl_Kep_1
      MOV     K2 C_Cyl_TF_SP.A_S_Cyl_Kep_2
      MOV     K2 C_Cyl_TF_SP.A_Status_XL_U
      MOV     K1 C_Cyl_TF_SP.A_S_Cyl_Tf
1979  LD=     Stp_TF_Fr K2
      MOV     K1 C_Cyl_TF_SP.A_S_Cyl_Kep_1
      MOV     K1 C_Cyl_TF_SP.A_S_Cyl_Kep_2
      MOV     K2 C_Cyl_TF_SP.A_Status_XL_U
      MOV     K1 C_Cyl_TF_SP.A_S_Cyl_Tf
2004  LD=     Stp_TF_Fr K3
      MOV     K1 C_Cyl_TF_SP.A_S_Cyl_Kep_1
      MOV     K1 C_Cyl_TF_SP.A_S_Cyl_Kep_2
      MOV     K1 C_Cyl_TF_SP.A_Status_XL_U
      MOV     K1 C_Cyl_TF_SP.A_S_Cyl_Tf
      MPS
      AND     M63
      SET     Skip_Heater
      MPP
      ANI     M63
      RST     Skip_Heater
2035  LD=     Stp_TF_Fr K4
      MOV     K1 C_Cyl_TF_SP.A_S_Cyl_Kep_1
      MOV     K1 C_Cyl_TF_SP.A_S_Cyl_Kep_2
      MOV     K1 C_Cyl_TF_SP.A_Status_XL_U
      MOV     K2 C_Cyl_TF_SP.A_S_Cyl_Tf
      AND     M72
      AND     M60
      OUT     D_Noti_Ex_Ep K10
2063  LD      D_Noti_Ex_Ep
      OUT     Ex_Ep_Frame
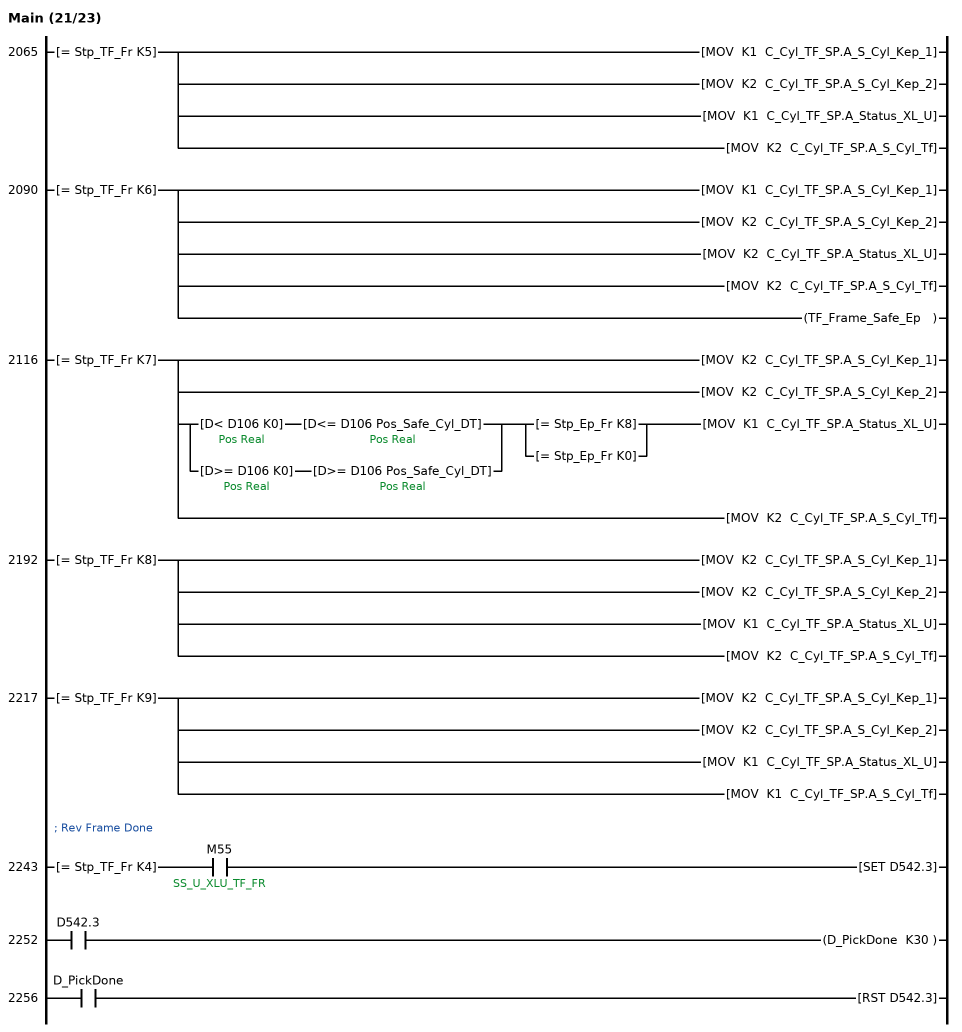
2065  LD=     Stp_TF_Fr K5
      MOV     K1 C_Cyl_TF_SP.A_S_Cyl_Kep_1
      MOV     K2 C_Cyl_TF_SP.A_S_Cyl_Kep_2
      MOV     K1 C_Cyl_TF_SP.A_Status_XL_U
      MOV     K2 C_Cyl_TF_SP.A_S_Cyl_Tf
2090  LD=     Stp_TF_Fr K6
      MOV     K1 C_Cyl_TF_SP.A_S_Cyl_Kep_1
      MOV     K2 C_Cyl_TF_SP.A_S_Cyl_Kep_2
      MOV     K2 C_Cyl_TF_SP.A_Status_XL_U
      MOV     K2 C_Cyl_TF_SP.A_S_Cyl_Tf
      OUT     TF_Frame_Safe_Ep
2116  LD=     Stp_TF_Fr K7
      MOV     K2 C_Cyl_TF_SP.A_S_Cyl_Kep_1
      MOV     K2 C_Cyl_TF_SP.A_S_Cyl_Kep_2
      MPS
      LDD<    D106 K0  ; Pos Real
      ANDD<=  D106 Pos_Safe_Cyl_DT  ; Pos Real
      LDD>=   D106 K0  ; Pos Real
      ANDD>=  D106 Pos_Safe_Cyl_DT  ; Pos Real
      ORB
      ANB
      LD=     Stp_Ep_Fr K8
      OR=     Stp_Ep_Fr K0
      ANB
      MOV     K1 C_Cyl_TF_SP.A_Status_XL_U
      MPP
      MOV     K2 C_Cyl_TF_SP.A_S_Cyl_Tf
2192  LD=     Stp_TF_Fr K8
      MOV     K2 C_Cyl_TF_SP.A_S_Cyl_Kep_1
      MOV     K2 C_Cyl_TF_SP.A_S_Cyl_Kep_2
      MOV     K1 C_Cyl_TF_SP.A_Status_XL_U
      MOV     K2 C_Cyl_TF_SP.A_S_Cyl_Tf
2217  LD=     Stp_TF_Fr K9
      MOV     K2 C_Cyl_TF_SP.A_S_Cyl_Kep_1
      MOV     K2 C_Cyl_TF_SP.A_S_Cyl_Kep_2
      MOV     K1 C_Cyl_TF_SP.A_Status_XL_U
      MOV     K1 C_Cyl_TF_SP.A_S_Cyl_Tf
; Rev Frame Done
2243  LD=     Stp_TF_Fr K4
      AND     M55  ; SS_U_XLU_TF_FR
      SET     D542.3
2252  LD      D542.3
      OUT     D_PickDone K30
2256  LD      D_PickDone
      RST     D542.3
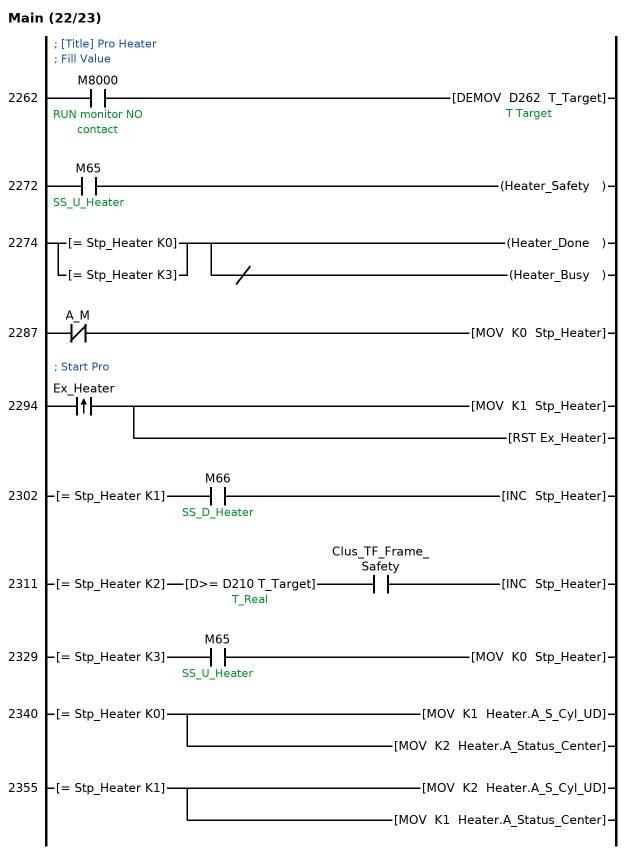
; [Title] Pro Heater
; Fill Value
2262  LD      M8000  ; RUN monitor NO contact
      DEMOV   D262 T_Target  ; T Target
2272  LD      M65  ; SS_U_Heater
      OUT     Heater_Safety
2274  LD=     Stp_Heater K0
      OR=     Stp_Heater K3
      OUT     Heater_Done
      INV
      OUT     Heater_Busy
2287  LDI     A_M
      MOV     K0 Stp_Heater
; Start Pro
2294  LDP     Ex_Heater
      MOV     K1 Stp_Heater
      RST     Ex_Heater
2302  LD=     Stp_Heater K1
      AND     M66  ; SS_D_Heater
      INC     Stp_Heater
2311  LD=     Stp_Heater K2
      ANDD>=  D210 T_Target  ; T_Real
      AND     Clus_TF_Frame_Safety
      INC     Stp_Heater
2329  LD=     Stp_Heater K3
      AND     M65  ; SS_U_Heater
      MOV     K0 Stp_Heater
2340  LD=     Stp_Heater K0
      MOV     K1 Heater.A_S_Cyl_UD
      MOV     K2 Heater.A_Status_Center
2355  LD=     Stp_Heater K1
      MOV     K2 Heater.A_S_Cyl_UD
      MOV     K1 Heater.A_Status_Center
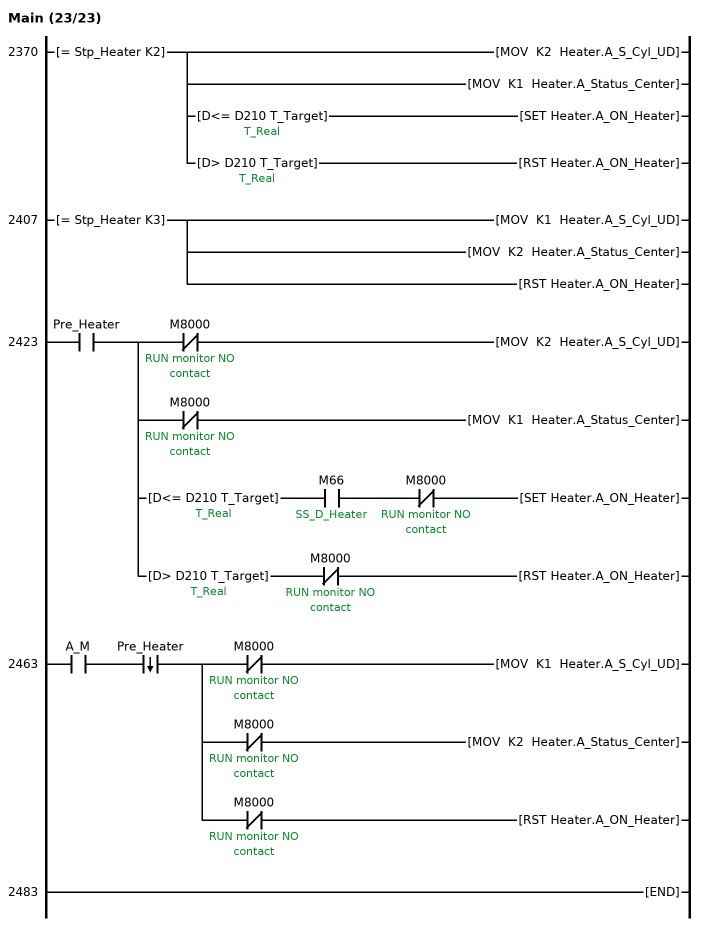
2370  LD=     Stp_Heater K2
      MOV     K2 Heater.A_S_Cyl_UD
      MOV     K1 Heater.A_Status_Center
      MPS
      ANDD<=  D210 T_Target  ; T_Real
      SET     Heater.A_ON_Heater
      MPP
      ANDD>   D210 T_Target  ; T_Real
      RST     Heater.A_ON_Heater
2407  LD=     Stp_Heater K3
      MOV     K1 Heater.A_S_Cyl_UD
      MOV     K2 Heater.A_Status_Center
      RST     Heater.A_ON_Heater
2423  LD      Pre_Heater
      MPS
      ANI     M8000  ; RUN monitor NO contact
      MOV     K2 Heater.A_S_Cyl_UD
      MRD
      ANI     M8000  ; RUN monitor NO contact
      MOV     K1 Heater.A_Status_Center
      MRD
      ANDD<=  D210 T_Target  ; T_Real
      AND     M66  ; SS_D_Heater
      ANI     M8000  ; RUN monitor NO contact
      SET     Heater.A_ON_Heater
      MPP
      ANDD>   D210 T_Target  ; T_Real
      ANI     M8000  ; RUN monitor NO contact
      RST     Heater.A_ON_Heater
2463  LD      A_M
      ANDF    Pre_Heater
      MPS
      ANI     M8000  ; RUN monitor NO contact
      MOV     K1 Heater.A_S_Cyl_UD
      MRD
      ANI     M8000  ; RUN monitor NO contact
      MOV     K2 Heater.A_Status_Center
      MPP
      ANI     M8000  ; RUN monitor NO contact
      RST     Heater.A_ON_Heater
2483  END
END_PROGRAM

FUNCTION_BLOCK Conv_TF_J
VAR_INPUT
  AM : BOOL;
  EMG : BOOL;
END_VAR
VAR_OUTPUT
  Org_Cyl_Keo : BOOL;
  Tf_Cyl_Keo : BOOL;
  Cyl_U_Jig : BOOL;
  Cyl_D_Jig : BOOL;
  R_FWD : BOOL;
  R_REV : BOOL;
END_VAR
VAR
  D_Rev_Jig : TIMER;
  T_L_R_A : TIMER;
END_VAR
VAR_INPUT
  I_M_FWD : BOOL;
  I_M_REV : BOOL;
  I_M_Stop : BOOL;
  I_M_U : BOOL;
  I_M_D : BOOL;
  I_M_Cyl_Org : BOOL;
  I_M_Cyl_Tf : BOOL;
  A_S_Cyl_UD : INT;
  A_S_Cyl_Tf : INT;
END_VAR
VAR
  A_FWD : BOOL;
  A_REV : BOOL;
  M_S_Cyl_UD : INT;
  M_FWD : BOOL;
  M_REV : BOOL;
  M_U : BOOL;
  A_U : BOOL;
  M_D : BOOL;
  A_D : BOOL;
  M_S_Cyl_Tf : INT;
  M_Cyl_Org : BOOL;
  M_XL_Tf : BOOL;
  A_XL_Tf : BOOL;
END_VAR
VAR_INPUT
  A_S_Conv : INT;
END_VAR
VAR
  A_Cyl_Org : BOOL;
END_VAR
VAR_INPUT
  L_C : BOOL;
  ORG : BOOL;
END_VAR
VAR_OUTPUT
  S_Org : BOOL;
END_VAR
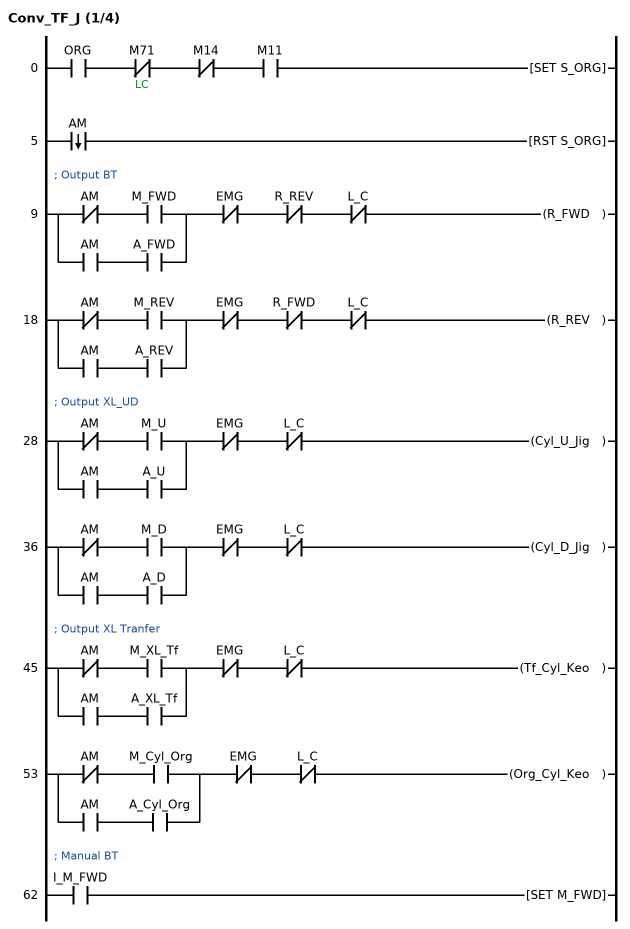
0     LD      ORG
      ANI     M71  ; LC
      ANI     M14
      AND     M11
      SET     S_ORG
5     LDF     AM
      RST     S_ORG
; Output BT
9     LDI     AM
      AND     M_FWD
      LD      AM
      AND     A_FWD
      ORB
      ANI     EMG
      ANI     R_REV
      ANI     L_C
      OUT     R_FWD
18    LDI     AM
      AND     M_REV
      LD      AM
      AND     A_REV
      ORB
      ANI     EMG
      ANI     R_FWD
      ANI     L_C
      OUT     R_REV
; Output XL_UD
28    LDI     AM
      AND     M_U
      LD      AM
      AND     A_U
      ORB
      ANI     EMG
      ANI     L_C
      OUT     Cyl_U_Jig
36    LDI     AM
      AND     M_D
      LD      AM
      AND     A_D
      ORB
      ANI     EMG
      ANI     L_C
      OUT     Cyl_D_Jig
; Output XL Tranfer
45    LDI     AM
      AND     M_XL_Tf
      LD      AM
      AND     A_XL_Tf
      ORB
      ANI     EMG
      ANI     L_C
      OUT     Tf_Cyl_Keo
53    LDI     AM
      AND     M_Cyl_Org
      LD      AM
      AND     A_Cyl_Org
      ORB
      ANI     EMG
      ANI     L_C
      OUT     Org_Cyl_Keo
; Manual BT
62    LD      I_M_FWD
      SET     M_FWD
